{attribute 'qualified_only'}
{attribute 'strict'}
TYPE E_IoDevice_ConnectionType :
(
    None := 0,              // the connection state is ignored (always FALSE)
	Strict := 1,            // the connection state can never vary 
    Timed := 2              // the connection is OFF if the timeout is violated
);
END_TYPE

(* stored: Version 1.1.0.1, ProductVersion 3.1.4024.9
   DUT E_IoDevice_ConnectionType: Id {6ea74376-0680-4dae-ac71-c40e62f0a732} *)
